(* Logix 5000 project; controller Tekno_ASRS vendor 1 type 14 code 147 rev 20.11; software revision 20.01; part 4 of 4 *)
(* tags used below, declared in another part *)
   AutoMode : BOOL;
   AAxis : AXIS_CIP_DRIVE;
   AAxisMAM : MOTION_INSTRUCTION;
   AAxisMove : BOOL;
   ABGrid : Position[100,20];
   ACompare : REAL;
   AftAreaRest : ALIAS FOR ShuttleIO:8:O.Pt05Data;
   AftAreaScanner : DCI_STOP;
   AftAreaZn1 : ALIAS FOR ShuttleIO:8:O.Pt07Data;
   AftAreaZn4 : ALIAS FOR ShuttleIO:8:O.Pt06Data;
   AftEndZn : BOOL;
   AGVDP : BOOL;
   AGVLightCurtains : DCI_STOP;
   AGVPU : BOOL;
   APos : REAL;
   AReq : DINT;
   ASRSEnable : BOOL;
   AutoConfig : Configuration;
   AxisEnabled : BOOL;
   BAxis : AXIS_CIP_DRIVE;
   BAxisMAM : MOTION_INSTRUCTION;
   BAxisMove : BOOL;
   BCompare : REAL;
   BlowerTm : TIMER;
   BPos : REAL;
   BReq : DINT;
   CommandReq : DINT;
   Configuration : Configuration;
   CReq : DINT;
   CurrentTask : Task;
   DepositReq : BOOL;
   DisableScanners : BOOL;
   DrivesOn : BOOL;
   EStop_SafetyGate : DCI_STOP;
   FootSwitch : ALIAS FOR ShuttleIO:9:I.Pt04Data;
   ForeAreaRst : ALIAS FOR ShuttleIO:8:O.Pt00Data;
   ForeAreaScanner : DCI_STOP;
   ForeAreaZn1 : ALIAS FOR ShuttleIO:8:O.Pt02Data;
   ForeAreaZn4 : ALIAS FOR ShuttleIO:8:O.Pt03Data;
   FwdEndZn : BOOL;
   GZReset : BOOL;
   HighSpdFwd : BOOL;
   HighSpdRev : BOOL;
   JogAct : BOOL;
   LiftStrnOK : BOOL;
   LightCur1 : ALIAS FOR StationaryIO:7:I.Pt06Data;
   LightCur2 : ALIAS FOR StationaryIO:7:I.Pt07Data;
   LightCurEN : ALIAS FOR StationaryIO:6:O.Pt07Data;
   ManConfig : Configuration;
   ManGateClosed : ALIAS FOR ShuttleIO:9:I.Pt02Data;
   MasterReset : BOOL;
   MoveRequested : BOOL;
   OperatorDN : BOOL;
   PalmButtonLeft : ALIAS FOR ShuttleIO:9:I.Pt07Data;
   PalmButtonRight : ALIAS FOR ShuttleIO:9:I.Pt06Data;
   PalmButtons : DCI_STOP;
   PDSimTmr : TIMER;
   ProxPwr : ALIAS FOR StationaryIO:6:O.Pt00Data;
   ResetSafety : BOOL;
   SafetyGate1 : ALIAS FOR StationaryIO:7:I.Pt00Data;
   SafetyGate2 : ALIAS FOR StationaryIO:7:I.Pt01Data;
   SafetyLaserAft1 : ALIAS FOR ShuttleIO:7:I.Pt04Data;
   SafetyLaserAft2 : ALIAS FOR ShuttleIO:7:I.Pt05Data;
   SafetyLaserFore1 : ALIAS FOR ShuttleIO:7:I.Pt00Data;
   SafetyLaserFore2 : ALIAS FOR ShuttleIO:7:I.Pt01Data;
   SafetyResetOns : BOOL;
   StationaryFault : BOOL;
   StationaryHorn : BOOL;
   StationaryManOn : BOOL;
   StationaryRun : BOOL;
   StationaryWarn : BOOL;
   Sts_ASRS_InputsOk : BOOL;
   TaskFIFO : CONTROL;
   TaskFile : Task[100];
   TaskInProcess : BOOL;
   UnBindInProc : BOOL;
   UnBindMotnInProc : BOOL;
   VFDReset : ALIAS FOR ShuttleIO:6:O.Pt00Data;
   XAccuracy : REAL;
   XAxisVFDSS01 : ALIAS FOR ShuttleIO:6:O.Pt04Data;
   XAxisVFDSS02 : ALIAS FOR ShuttleIO:6:O.Pt05Data;
   XHighLimit : REAL;
   XLowLimit : REAL;
   XStrain : Strain;
   XStrainLeftMax : DINT;
   XStrainLeftMin : DINT;
   XStrainRightMax : DINT;
   XStrainRightMin : DINT;
   ZAccuracy : REAL;
   ZADisengage : BOOL;
   ZAftLeftOK : BOOL;
   ZAftRightOK : BOOL;
   ZAftStCalMode : ALIAS FOR ShuttleIO:4:O.Data[0].0;
   ZAftStLftSignRun : ALIAS FOR ShuttleIO:4:I.Data[7].7;
   ZAftStrain : Strain;
   ZAftStrainLeftMax : DINT;
   ZAftStrainLeftMin : DINT;
   ZAftStrainRightMax : DINT;
   ZAftStrainRightMin : DINT;
   ZAftStRtSignRun : ALIAS FOR ShuttleIO:4:I.Data[11].7;
   ZAftStRunMode : ALIAS FOR ShuttleIO:4:O.Data[0].1;
   ZALftTempDint1 : DINT;
   ZALftTempDint2 : DINT;
   ZALftTempFloat1 : REAL;
   ZALftTempFloat2 : REAL;
   ZALftTempFloat3 : REAL;
   ZARgtTempDint1 : DINT;
   ZARgtTempDint2 : DINT;
   ZARgtTempFloat1 : REAL;
   ZARgtTempFloat2 : REAL;
   ZARgtTempFloat3 : REAL;
   ZAxisSafetyDisengage : BOOL;
   ZAxisSafetyLatches : ALIAS FOR ShuttleIO:6:O.Pt07Data;
   ZFLftTempDint1 : DINT;
   ZFLftTempDint2 : DINT;
   ZFLftTempFloat1 : REAL;
   ZFLftTempFloat2 : REAL;
   ZFLftTempFloat3 : REAL;
   ZForeLeftOK : BOOL;
   ZForeRightOK : BOOL;
   ZForeStCalMode : ALIAS FOR ShuttleIO:3:O.Data[0].0;
   ZForeStLftSignRun : ALIAS FOR ShuttleIO:3:I.Data[7].7;
   ZForeStrain : Strain;
   ZForeStrainLeftMax : DINT;
   ZForeStrainLeftMin : DINT;
   ZForeStrainRightMax : DINT;
   ZForeStrainRightMin : DINT;
   ZForeStRtSignRun : ALIAS FOR ShuttleIO:3:I.Data[11].7;
   ZForeStRunMode : ALIAS FOR ShuttleIO:3:O.Data[0].1;
   ZFRgtTempDint1 : DINT;
   ZFRgtTempDint2 : DINT;
   ZFRgtTempFloat1 : REAL;
   ZFRgtTempFloat2 : REAL;
   ZFRgtTempFloat3 : REAL;
   ZHighLimit : REAL;
   ZLBindTmr : TIMER;
   ZLFault : BOOL;
   ZLockMove : MOTION_INSTRUCTION;
   ZLowLimit : REAL;
   ZLProxOK : BOOL;
   ZLReqPosition : REAL;
   ZLRetryDelay : TIMER;
   ZStrainHigh : DINT;
   ZStrainLow : DINT;
(* MainProgram, continued *)

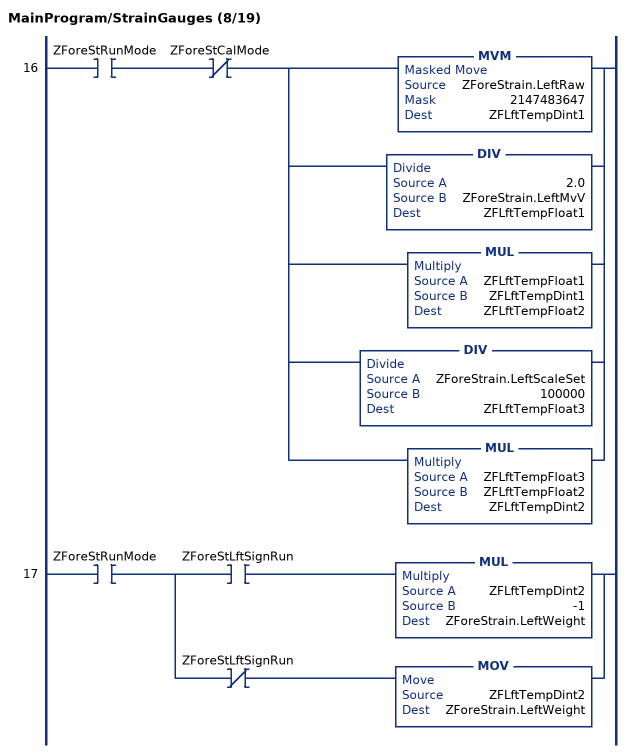
   [picture p48: MainProgram/StrainGauges rungs 16-17]
   16: XIC(ZForeStRunMode)XIO(ZForeStCalMode)[MVM(ZForeStrain.LeftRaw,2147483647,ZFLftTempDint1) ,DIV(2.0,ZForeStrain.LeftMvV,ZFLftTempFloat1) ,MUL(ZFLftTempFloat1,ZFLftTempDint1,ZFLftTempFloat2) ,DIV(ZForeStrain.LeftScaleSet,100000,ZFLftTempFloat3) ,MUL(ZFLftTempFloat3,ZFLftTempFloat2,ZFLftTempDint2) ];
   17: XIC(ZForeStRunMode)[XIC(ZForeStLftSignRun) MUL(ZFLftTempDint2,-1,ZForeStrain.LeftWeight) ,XIO(ZForeStLftSignRun) MOV(ZFLftTempDint2,ZForeStrain.LeftWeight) ];
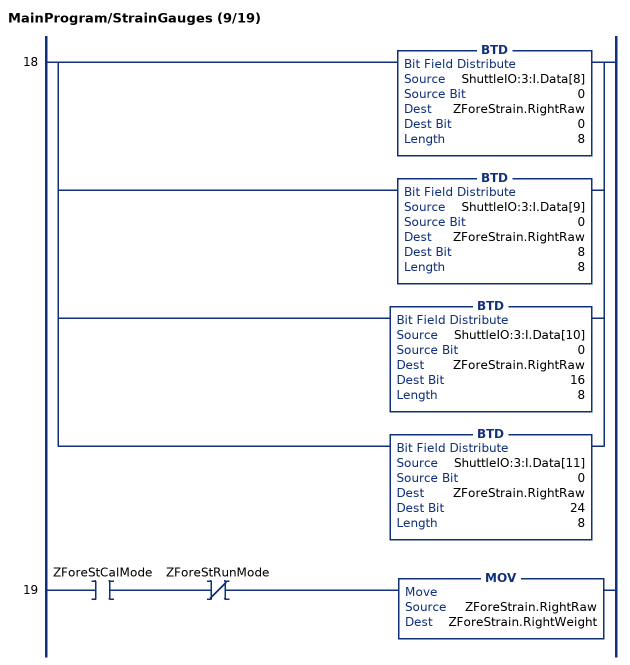
   18: [BTD(ShuttleIO:3:I.Data[8],0,ZForeStrain.RightRaw,0,8) ,BTD(ShuttleIO:3:I.Data[9],0,ZForeStrain.RightRaw,8,8) ,BTD(ShuttleIO:3:I.Data[10],0,ZForeStrain.RightRaw,16,8) ,BTD(ShuttleIO:3:I.Data[11],0,ZForeStrain.RightRaw,24,8) ];
   19: XIC(ZForeStCalMode)XIO(ZForeStRunMode)MOV(ZForeStrain.RightRaw,ZForeStrain.RightWeight);
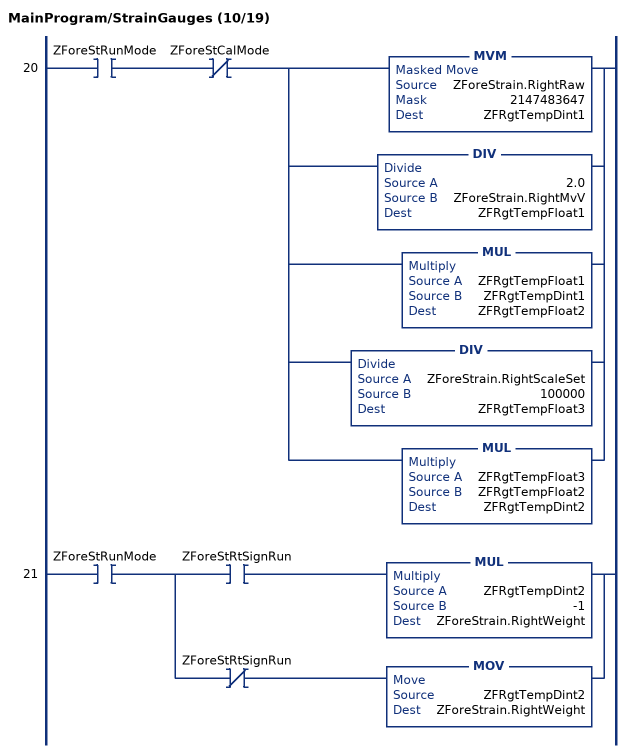
   20: XIC(ZForeStRunMode)XIO(ZForeStCalMode)[MVM(ZForeStrain.RightRaw,2147483647,ZFRgtTempDint1) ,DIV(2.0,ZForeStrain.RightMvV,ZFRgtTempFloat1) ,MUL(ZFRgtTempFloat1,ZFRgtTempDint1,ZFRgtTempFloat2) ,DIV(ZForeStrain.RightScaleSet,100000,ZFRgtTempFloat3) ,MUL(ZFRgtTempFloat3,ZFRgtTempFloat2,ZFRgtTempDint2) ];
   21: XIC(ZForeStRunMode)[XIC(ZForeStRtSignRun) MUL(ZFRgtTempDint2,-1,ZForeStrain.RightWeight) ,XIO(ZForeStRtSignRun) MOV(ZFRgtTempDint2,ZForeStrain.RightWeight) ];
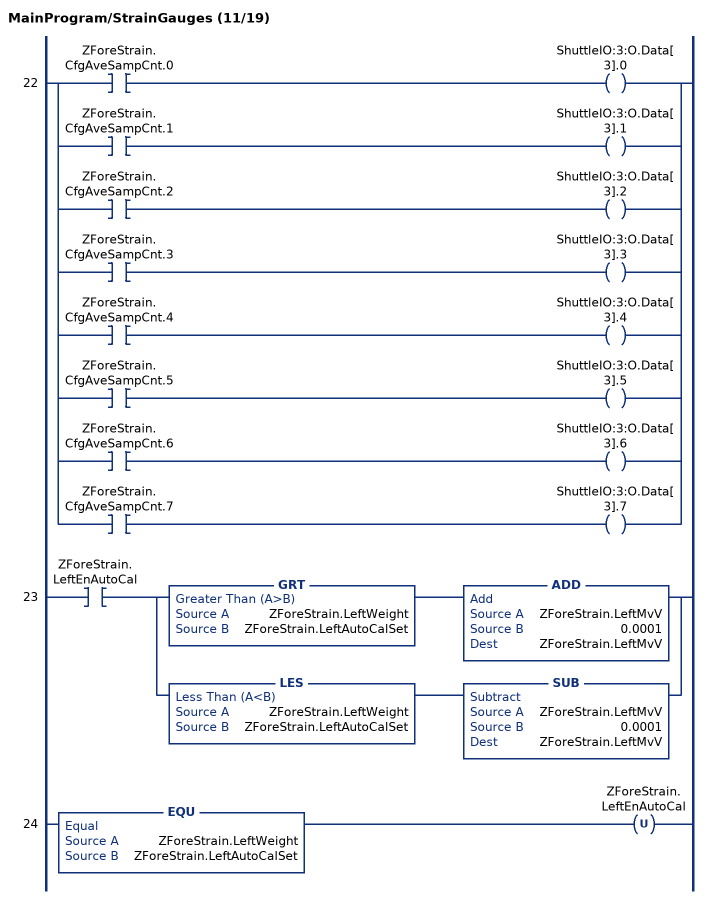
   22: [XIC(ZForeStrain.CfgAveSampCnt.0) OTE(ShuttleIO:3:O.Data[3].0) ,XIC(ZForeStrain.CfgAveSampCnt.1) OTE(ShuttleIO:3:O.Data[3].1) ,XIC(ZForeStrain.CfgAveSampCnt.2) OTE(ShuttleIO:3:O.Data[3].2) ,XIC(ZForeStrain.CfgAveSampCnt.3) OTE(ShuttleIO:3:O.Data[3].3) ,XIC(ZForeStrain.CfgAveSampCnt.4) OTE(ShuttleIO:3:O.Data[3].4) ,XIC(ZForeStrain.CfgAveSampCnt.5) OTE(ShuttleIO:3:O.Data[3].5) ,XIC(ZForeStrain.CfgAveSampCnt.6) OTE(ShuttleIO:3:O.Data[3].6) ,XIC(ZForeStrain.CfgAveSampCnt.7) OTE(ShuttleIO:3:O.Data[3].7) ];
   23: XIC(ZForeStrain.LeftEnAutoCal)[GRT(ZForeStrain.LeftWeight,ZForeStrain.LeftAutoCalSet) ADD(ZForeStrain.LeftMvV,0.0001,ZForeStrain.LeftMvV) ,LES(ZForeStrain.LeftWeight,ZForeStrain.LeftAutoCalSet) SUB(ZForeStrain.LeftMvV,0.0001,ZForeStrain.LeftMvV) ];
   24: EQU(ZForeStrain.LeftWeight,ZForeStrain.LeftAutoCalSet)OTU(ZForeStrain.LeftEnAutoCal);
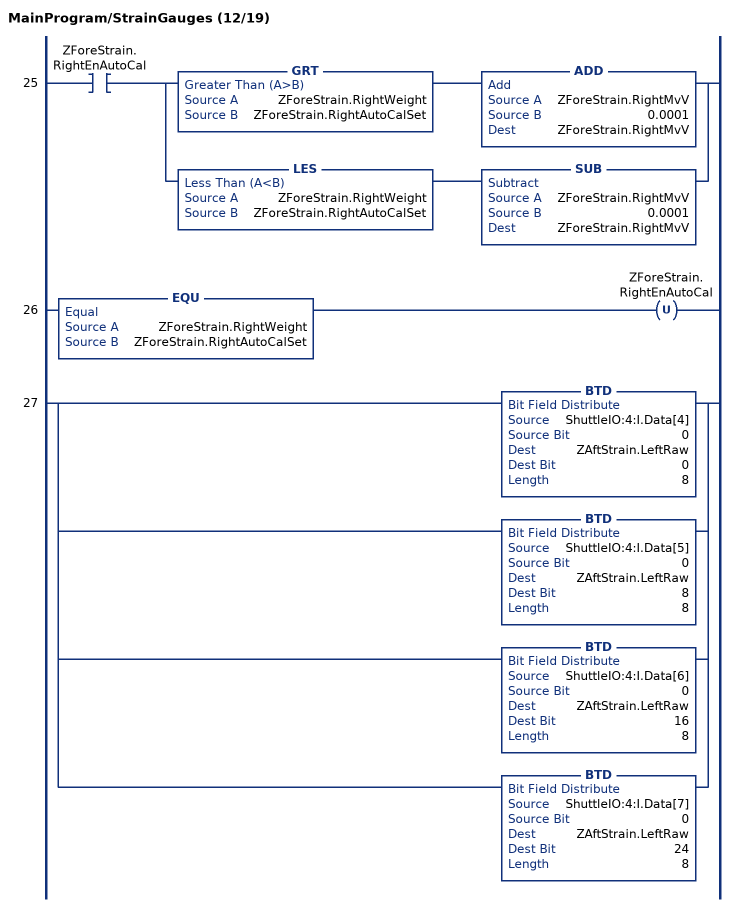
   25: XIC(ZForeStrain.RightEnAutoCal)[GRT(ZForeStrain.RightWeight,ZForeStrain.RightAutoCalSet) ADD(ZForeStrain.RightMvV,0.0001,ZForeStrain.RightMvV) ,LES(ZForeStrain.RightWeight,ZForeStrain.RightAutoCalSet) SUB(ZForeStrain.RightMvV,0.0001,ZForeStrain.RightMvV) ];
   26: EQU(ZForeStrain.RightWeight,ZForeStrain.RightAutoCalSet)OTU(ZForeStrain.RightEnAutoCal);
   27: [BTD(ShuttleIO:4:I.Data[4],0,ZAftStrain.LeftRaw,0,8) ,BTD(ShuttleIO:4:I.Data[5],0,ZAftStrain.LeftRaw,8,8) ,BTD(ShuttleIO:4:I.Data[6],0,ZAftStrain.LeftRaw,16,8) ,BTD(ShuttleIO:4:I.Data[7],0,ZAftStrain.LeftRaw,24,8) ];
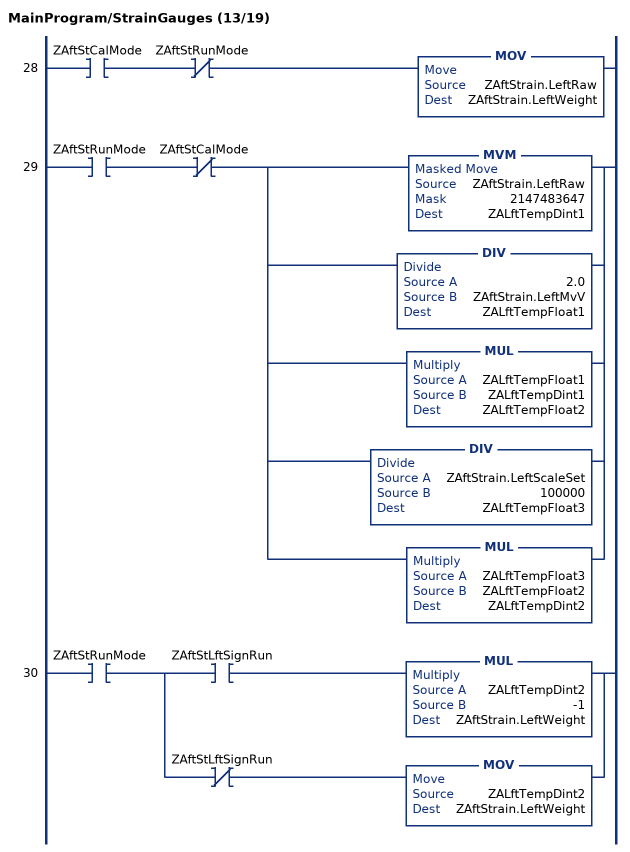
   28: XIC(ZAftStCalMode)XIO(ZAftStRunMode)MOV(ZAftStrain.LeftRaw,ZAftStrain.LeftWeight);
   29: XIC(ZAftStRunMode)XIO(ZAftStCalMode)[MVM(ZAftStrain.LeftRaw,2147483647,ZALftTempDint1) ,DIV(2.0,ZAftStrain.LeftMvV,ZALftTempFloat1) ,MUL(ZALftTempFloat1,ZALftTempDint1,ZALftTempFloat2) ,DIV(ZAftStrain.LeftScaleSet,100000,ZALftTempFloat3) ,MUL(ZALftTempFloat3,ZALftTempFloat2,ZALftTempDint2) ];
   30: XIC(ZAftStRunMode)[XIC(ZAftStLftSignRun) MUL(ZALftTempDint2,-1,ZAftStrain.LeftWeight) ,XIO(ZAftStLftSignRun) MOV(ZALftTempDint2,ZAftStrain.LeftWeight) ];
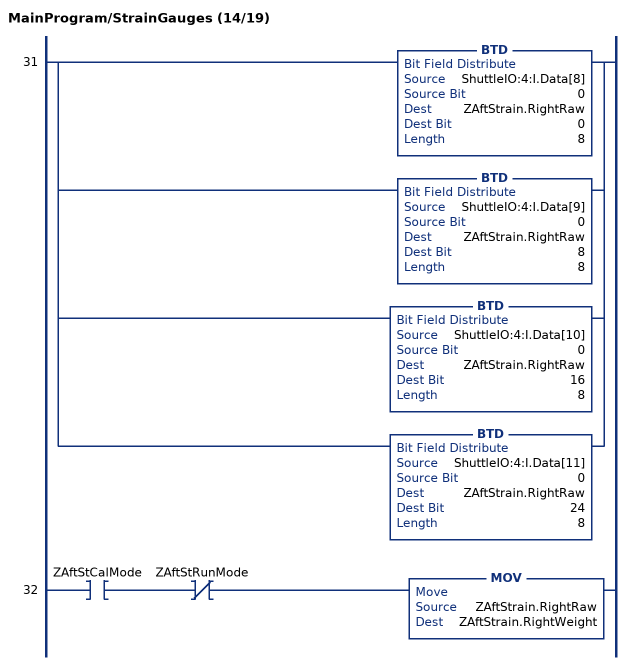
   31: [BTD(ShuttleIO:4:I.Data[8],0,ZAftStrain.RightRaw,0,8) ,BTD(ShuttleIO:4:I.Data[9],0,ZAftStrain.RightRaw,8,8) ,BTD(ShuttleIO:4:I.Data[10],0,ZAftStrain.RightRaw,16,8) ,BTD(ShuttleIO:4:I.Data[11],0,ZAftStrain.RightRaw,24,8) ];
   32: XIC(ZAftStCalMode)XIO(ZAftStRunMode)MOV(ZAftStrain.RightRaw,ZAftStrain.RightWeight);
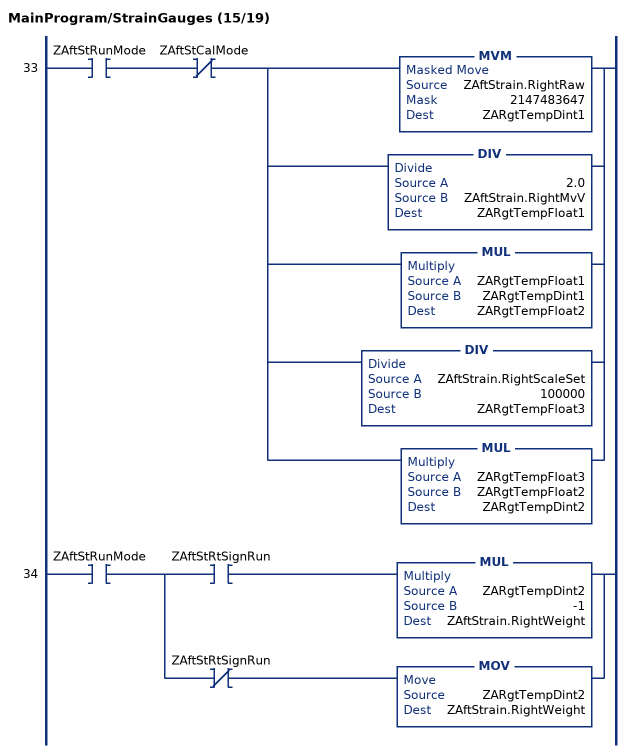
   33: XIC(ZAftStRunMode)XIO(ZAftStCalMode)[MVM(ZAftStrain.RightRaw,2147483647,ZARgtTempDint1) ,DIV(2.0,ZAftStrain.RightMvV,ZARgtTempFloat1) ,MUL(ZARgtTempFloat1,ZARgtTempDint1,ZARgtTempFloat2) ,DIV(ZAftStrain.RightScaleSet,100000,ZARgtTempFloat3) ,MUL(ZARgtTempFloat3,ZARgtTempFloat2,ZARgtTempDint2) ];
   34: XIC(ZAftStRunMode)[XIC(ZAftStRtSignRun) MUL(ZARgtTempDint2,-1,ZAftStrain.RightWeight) ,XIO(ZAftStRtSignRun) MOV(ZARgtTempDint2,ZAftStrain.RightWeight) ];
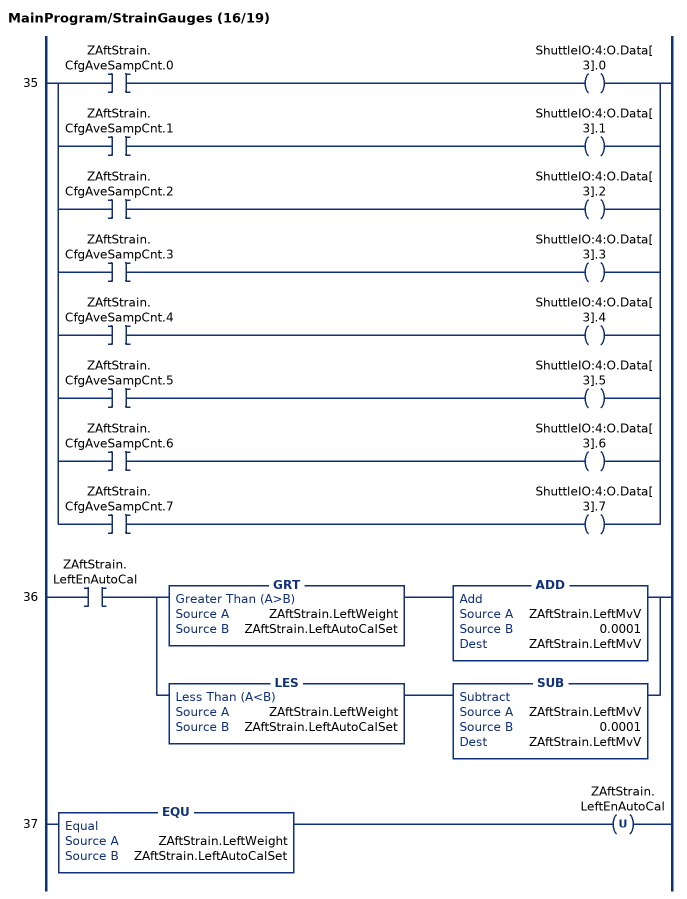
   35: [XIC(ZAftStrain.CfgAveSampCnt.0) OTE(ShuttleIO:4:O.Data[3].0) ,XIC(ZAftStrain.CfgAveSampCnt.1) OTE(ShuttleIO:4:O.Data[3].1) ,XIC(ZAftStrain.CfgAveSampCnt.2) OTE(ShuttleIO:4:O.Data[3].2) ,XIC(ZAftStrain.CfgAveSampCnt.3) OTE(ShuttleIO:4:O.Data[3].3) ,XIC(ZAftStrain.CfgAveSampCnt.4) OTE(ShuttleIO:4:O.Data[3].4) ,XIC(ZAftStrain.CfgAveSampCnt.5) OTE(ShuttleIO:4:O.Data[3].5) ,XIC(ZAftStrain.CfgAveSampCnt.6) OTE(ShuttleIO:4:O.Data[3].6) ,XIC(ZAftStrain.CfgAveSampCnt.7) OTE(ShuttleIO:4:O.Data[3].7) ];
   36: XIC(ZAftStrain.LeftEnAutoCal)[GRT(ZAftStrain.LeftWeight,ZAftStrain.LeftAutoCalSet) ADD(ZAftStrain.LeftMvV,0.0001,ZAftStrain.LeftMvV) ,LES(ZAftStrain.LeftWeight,ZAftStrain.LeftAutoCalSet) SUB(ZAftStrain.LeftMvV,0.0001,ZAftStrain.LeftMvV) ];
   37: EQU(ZAftStrain.LeftWeight,ZAftStrain.LeftAutoCalSet)OTU(ZAftStrain.LeftEnAutoCal);
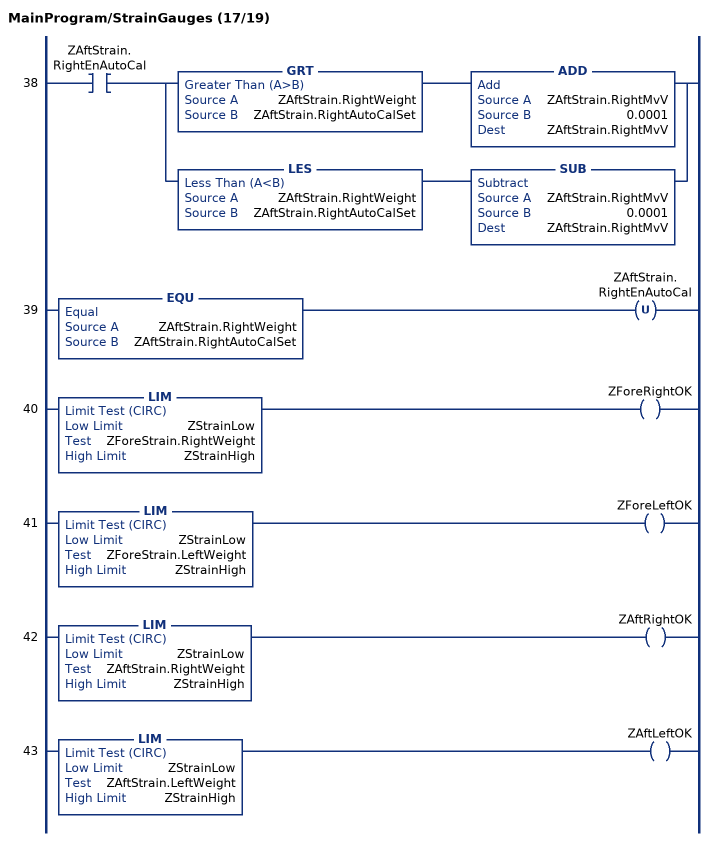
   38: XIC(ZAftStrain.RightEnAutoCal)[GRT(ZAftStrain.RightWeight,ZAftStrain.RightAutoCalSet) ADD(ZAftStrain.RightMvV,0.0001,ZAftStrain.RightMvV) ,LES(ZAftStrain.RightWeight,ZAftStrain.RightAutoCalSet) SUB(ZAftStrain.RightMvV,0.0001,ZAftStrain.RightMvV) ];
   39: EQU(ZAftStrain.RightWeight,ZAftStrain.RightAutoCalSet)OTU(ZAftStrain.RightEnAutoCal);
   40: LIM(ZStrainLow,ZForeStrain.RightWeight,ZStrainHigh)OTE(ZForeRightOK);
   41: LIM(ZStrainLow,ZForeStrain.LeftWeight,ZStrainHigh)OTE(ZForeLeftOK);
   42: LIM(ZStrainLow,ZAftStrain.RightWeight,ZStrainHigh)OTE(ZAftRightOK);
   43: LIM(ZStrainLow,ZAftStrain.LeftWeight,ZStrainHigh)OTE(ZAftLeftOK);
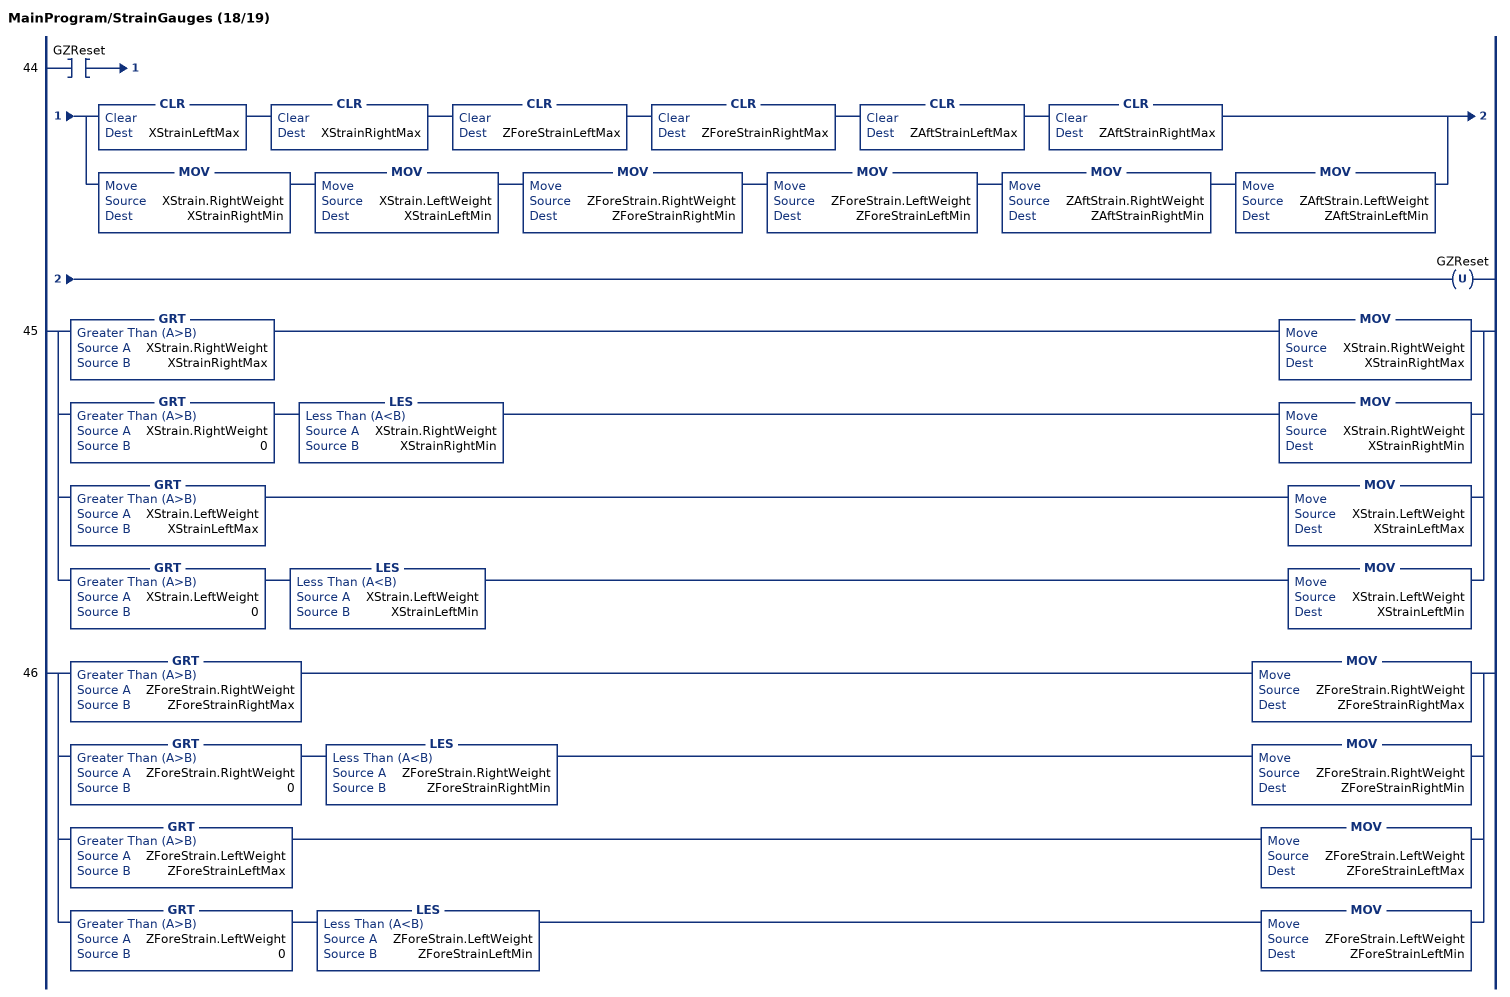
   44: XIC(GZReset)[CLR(XStrainLeftMax) CLR(XStrainRightMax) CLR(ZForeStrainLeftMax) CLR(ZForeStrainRightMax) CLR(ZAftStrainLeftMax) CLR(ZAftStrainRightMax) ,MOV(XStrain.RightWeight,XStrainRightMin) MOV(XStrain.LeftWeight,XStrainLeftMin) MOV(ZForeStrain.RightWeight,ZForeStrainRightMin) MOV(ZForeStrain.LeftWeight,ZForeStrainLeftMin) MOV(ZAftStrain.RightWeight,ZAftStrainRightMin) MOV(ZAftStrain.LeftWeight,ZAftStrainLeftMin) ]OTU(GZReset);
   45: [GRT(XStrain.RightWeight,XStrainRightMax) MOV(XStrain.RightWeight,XStrainRightMax) ,GRT(XStrain.RightWeight,0) LES(XStrain.RightWeight,XStrainRightMin) MOV(XStrain.RightWeight,XStrainRightMin) ,GRT(XStrain.LeftWeight,XStrainLeftMax) MOV(XStrain.LeftWeight,XStrainLeftMax) ,GRT(XStrain.LeftWeight,0) LES(XStrain.LeftWeight,XStrainLeftMin) MOV(XStrain.LeftWeight,XStrainLeftMin) ];
   46: [GRT(ZForeStrain.RightWeight,ZForeStrainRightMax) MOV(ZForeStrain.RightWeight,ZForeStrainRightMax) ,GRT(ZForeStrain.RightWeight,0) LES(ZForeStrain.RightWeight,ZForeStrainRightMin) MOV(ZForeStrain.RightWeight,ZForeStrainRightMin) ,GRT(ZForeStrain.LeftWeight,ZForeStrainLeftMax) MOV(ZForeStrain.LeftWeight,ZForeStrainLeftMax) ,GRT(ZForeStrain.LeftWeight,0) LES(ZForeStrain.LeftWeight,ZForeStrainLeftMin) MOV(ZForeStrain.LeftWeight,ZForeStrainLeftMin) ];
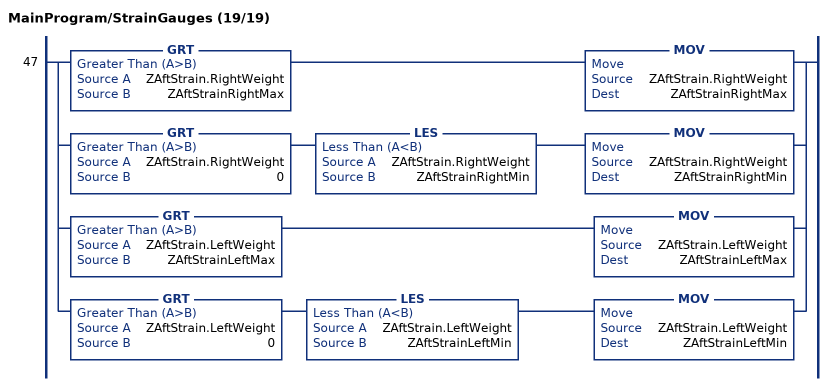
   47: [GRT(ZAftStrain.RightWeight,ZAftStrainRightMax) MOV(ZAftStrain.RightWeight,ZAftStrainRightMax) ,GRT(ZAftStrain.RightWeight,0) LES(ZAftStrain.RightWeight,ZAftStrainRightMin) MOV(ZAftStrain.RightWeight,ZAftStrainRightMin) ,GRT(ZAftStrain.LeftWeight,ZAftStrainLeftMax) MOV(ZAftStrain.LeftWeight,ZAftStrainLeftMax) ,GRT(ZAftStrain.LeftWeight,0) LES(ZAftStrain.LeftWeight,ZAftStrainLeftMin) MOV(ZAftStrain.LeftWeight,ZAftStrainLeftMin) ];
END_ROUTINE

ROUTINE Task_List_Processor   (* ladder *)
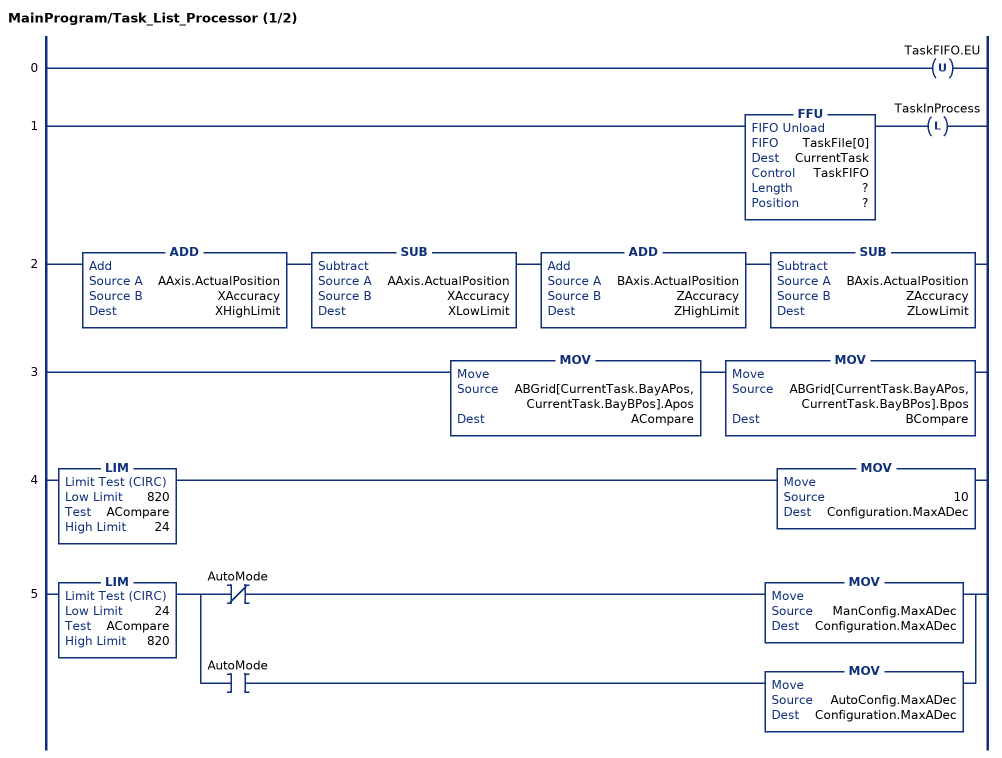
   0: OTU(TaskFIFO.EU);
   1: FFU(TaskFile[0],CurrentTask,TaskFIFO,?,?)OTL(TaskInProcess);
   2: ADD(AAxis.ActualPosition,XAccuracy,XHighLimit)SUB(AAxis.ActualPosition,XAccuracy,XLowLimit)ADD(BAxis.ActualPosition,ZAccuracy,ZHighLimit)SUB(BAxis.ActualPosition,ZAccuracy,ZLowLimit);
   3: MOV(ABGrid[CurrentTask.BayAPos,CurrentTask.BayBPos].Apos,ACompare)MOV(ABGrid[CurrentTask.BayAPos,CurrentTask.BayBPos].Bpos,BCompare);
   4: LIM(820,ACompare,24)MOV(10,Configuration.MaxADec);
   5: LIM(24,ACompare,820)[XIO(AutoMode) MOV(ManConfig.MaxADec,Configuration.MaxADec) ,XIC(AutoMode) MOV(AutoConfig.MaxADec,Configuration.MaxADec) ];
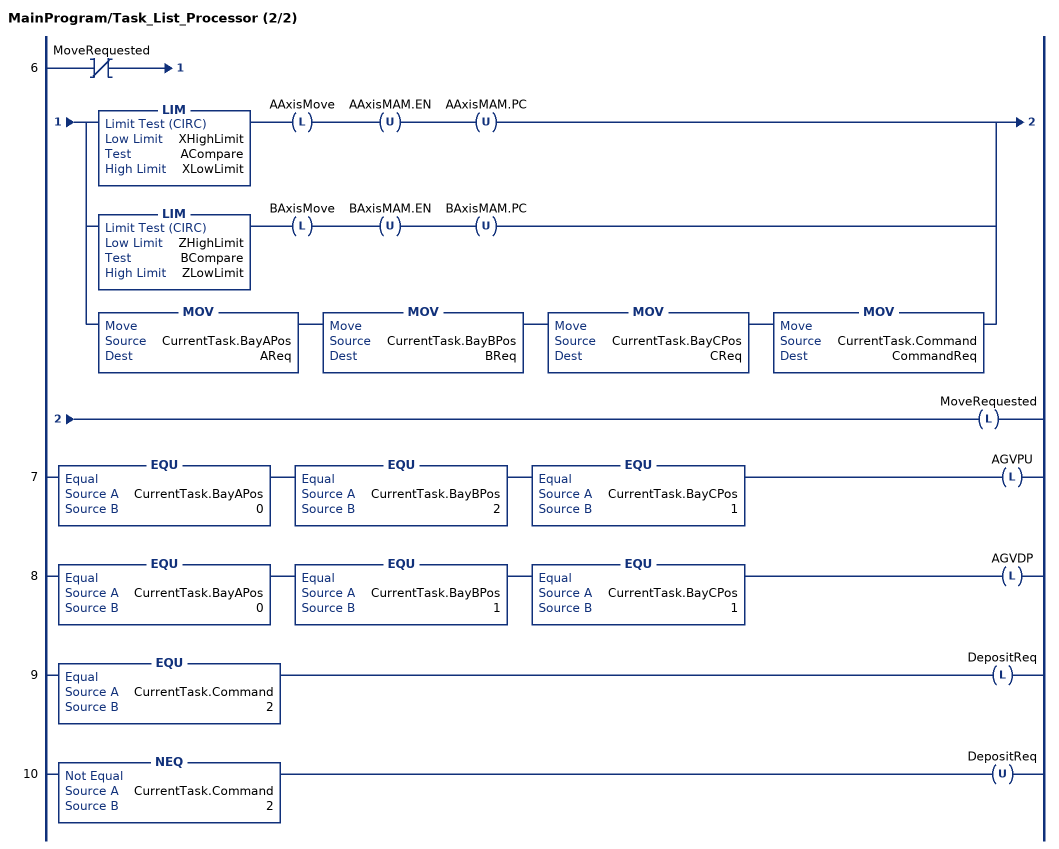
   6: XIO(MoveRequested)[LIM(XHighLimit,ACompare,XLowLimit) OTL(AAxisMove) OTU(AAxisMAM.EN) OTU(AAxisMAM.PC) ,LIM(ZHighLimit,BCompare,ZLowLimit) OTL(BAxisMove) OTU(BAxisMAM.EN) OTU(BAxisMAM.PC) ,MOV(CurrentTask.BayAPos,AReq) MOV(CurrentTask.BayBPos,BReq) MOV(CurrentTask.BayCPos,CReq) MOV(CurrentTask.Command,CommandReq) ]OTL(MoveRequested);
   7: EQU(CurrentTask.BayAPos,0)EQU(CurrentTask.BayBPos,2)EQU(CurrentTask.BayCPos,1)OTL(AGVPU);
   8: EQU(CurrentTask.BayAPos,0)EQU(CurrentTask.BayBPos,1)EQU(CurrentTask.BayCPos,1)OTL(AGVDP);
   9: EQU(CurrentTask.Command,2)OTL(DepositReq);
   10: NEQ(CurrentTask.Command,2)OTU(DepositReq);
END_ROUTINE

ROUTINE VisitPorD   (* ladder *)
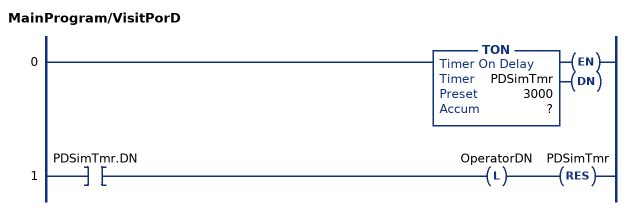
   0: TON(PDSimTmr,?,?);
   1: XIC(PDSimTmr.DN)OTL(OperatorDN)RES(PDSimTmr);
END_ROUTINE

ROUTINE ZLock_Release   (* ladder *)
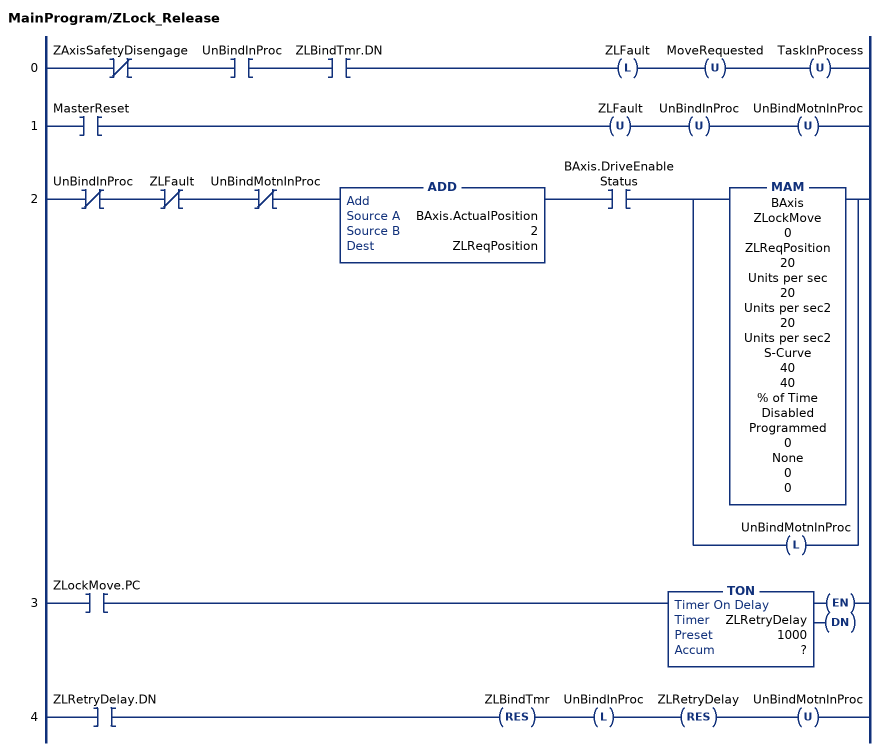
   0: XIO(ZAxisSafetyDisengage)XIC(UnBindInProc)XIC(ZLBindTmr.DN)OTL(ZLFault)OTU(MoveRequested)OTU(TaskInProcess);
   1: XIC(MasterReset)OTU(ZLFault)OTU(UnBindInProc)OTU(UnBindMotnInProc);
   2: XIO(UnBindInProc)XIO(ZLFault)XIO(UnBindMotnInProc)ADD(BAxis.ActualPosition,2,ZLReqPosition)XIC(BAxis.DriveEnableStatus)[MAM(BAxis,ZLockMove,0,ZLReqPosition,20,Units per sec,20,Units per sec2,20,Units per sec2,S-Curve,40,40,% of Time,Disabled,Programmed,0,None,0,0) ,OTL(UnBindMotnInProc) ];
   3: XIC(ZLockMove.PC)TON(ZLRetryDelay,?,?);
   4: XIC(ZLRetryDelay.DN)RES(ZLBindTmr)OTL(UnBindInProc)RES(ZLRetryDelay)OTU(UnBindMotnInProc);
END_ROUTINE
END_PROGRAM

PROGRAM SafetyProgram   (* main routine MainRoutine *)
VAR
   alkjdfl : BOOL;
   Lift : DINT;
   ljfalsj : BOOL;
END_VAR

ROUTINE MainRoutine   (* ladder *)
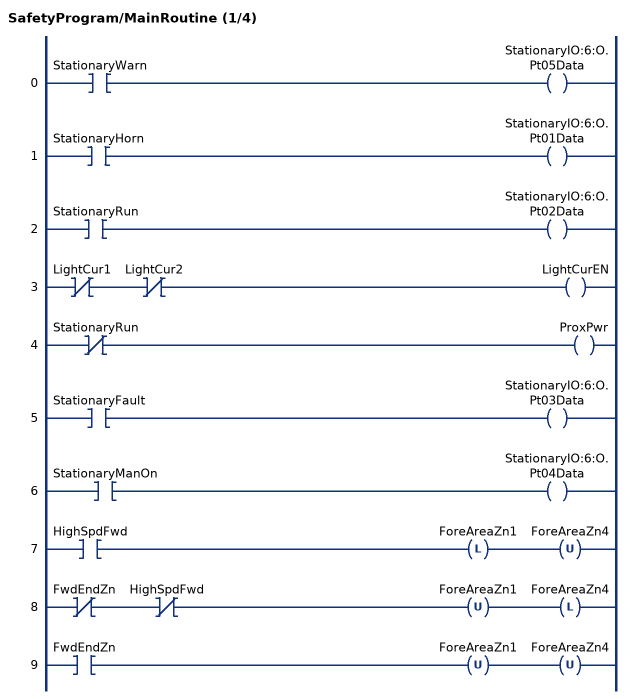
   0: XIC(StationaryWarn)OTE(StationaryIO:6:O.Pt05Data);
   1: XIC(StationaryHorn)OTE(StationaryIO:6:O.Pt01Data);
   2: XIC(StationaryRun)OTE(StationaryIO:6:O.Pt02Data);
   3: XIO(LightCur1)XIO(LightCur2)OTE(LightCurEN);
   4: XIO(StationaryRun)OTE(ProxPwr);
   5: XIC(StationaryFault)OTE(StationaryIO:6:O.Pt03Data);
   6: XIC(StationaryManOn)OTE(StationaryIO:6:O.Pt04Data);
   7: XIC(HighSpdFwd)OTL(ForeAreaZn1)OTU(ForeAreaZn4);
   8: XIO(FwdEndZn)XIO(HighSpdFwd)OTU(ForeAreaZn1)OTL(ForeAreaZn4);
   9: XIC(FwdEndZn)OTU(ForeAreaZn1)OTU(ForeAreaZn4);
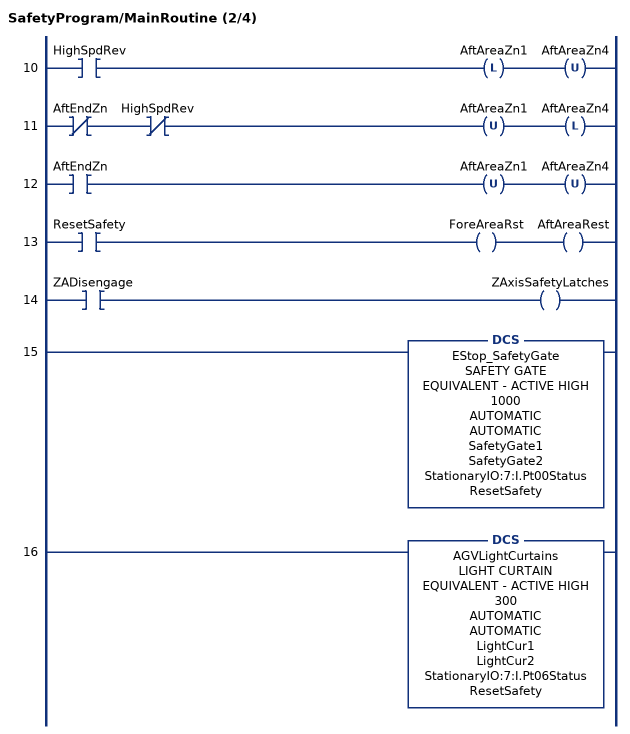
   10: XIC(HighSpdRev)OTL(AftAreaZn1)OTU(AftAreaZn4);
   11: XIO(AftEndZn)XIO(HighSpdRev)OTU(AftAreaZn1)OTL(AftAreaZn4);
   12: XIC(AftEndZn)OTU(AftAreaZn1)OTU(AftAreaZn4);
   13: XIC(ResetSafety)OTE(ForeAreaRst)OTE(AftAreaRest);
   14: XIC(ZADisengage)OTE(ZAxisSafetyLatches);
   15: DCS(EStop_SafetyGate,SAFETY GATE,EQUIVALENT - ACTIVE HIGH,1000,AUTOMATIC,AUTOMATIC,SafetyGate1,SafetyGate2,StationaryIO:7:I.Pt00Status,ResetSafety);
   16: DCS(AGVLightCurtains,LIGHT CURTAIN,EQUIVALENT - ACTIVE HIGH,300,AUTOMATIC,AUTOMATIC,LightCur1,LightCur2,StationaryIO:7:I.Pt06Status,ResetSafety);
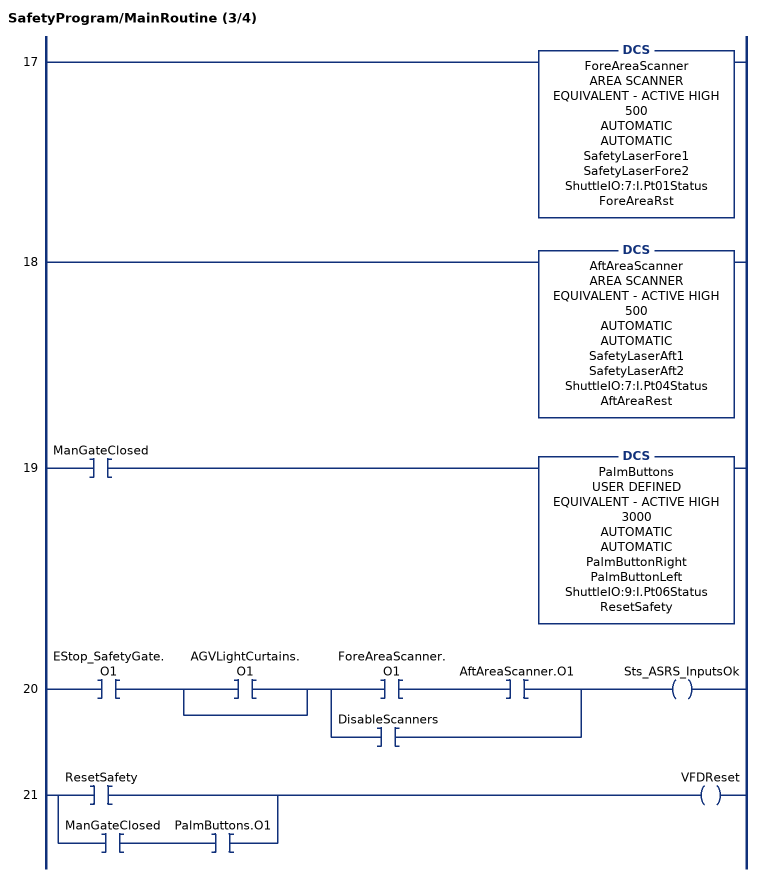
   17: DCS(ForeAreaScanner,AREA SCANNER,EQUIVALENT - ACTIVE HIGH,500,AUTOMATIC,AUTOMATIC,SafetyLaserFore1,SafetyLaserFore2,ShuttleIO:7:I.Pt01Status,ForeAreaRst);
   18: DCS(AftAreaScanner,AREA SCANNER,EQUIVALENT - ACTIVE HIGH,500,AUTOMATIC,AUTOMATIC,SafetyLaserAft1,SafetyLaserAft2,ShuttleIO:7:I.Pt04Status,AftAreaRest);
   19: XIC(ManGateClosed)DCS(PalmButtons,USER DEFINED,EQUIVALENT - ACTIVE HIGH,3000,AUTOMATIC,AUTOMATIC,PalmButtonRight,PalmButtonLeft,ShuttleIO:9:I.Pt06Status,ResetSafety);
   20: XIC(EStop_SafetyGate.O1)[XIC(AGVLightCurtains.O1) ,][XIC(ForeAreaScanner.O1) XIC(AftAreaScanner.O1) ,XIC(DisableScanners) ]OTE(Sts_ASRS_InputsOk);
   21: [XIC(ResetSafety) ,XIC(ManGateClosed) XIC(PalmButtons.O1) ]OTE(VFDReset);
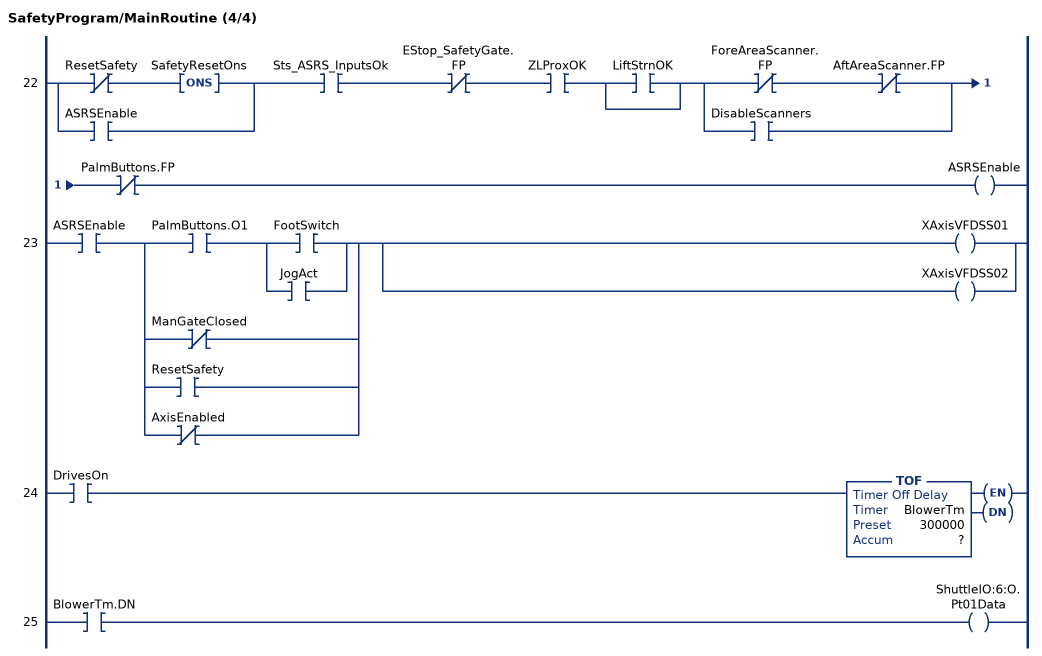
   22: [XIO(ResetSafety) ONS(SafetyResetOns) ,XIC(ASRSEnable) ]XIC(Sts_ASRS_InputsOk)XIO(EStop_SafetyGate.FP)XIC(ZLProxOK)[XIC(LiftStrnOK) ,][XIO(ForeAreaScanner.FP) XIO(AftAreaScanner.FP) ,XIC(DisableScanners) ]XIO(PalmButtons.FP)OTE(ASRSEnable);
   23: XIC(ASRSEnable)[XIC(PalmButtons.O1) [XIC(FootSwitch) ,XIC(JogAct) ] ,XIO(ManGateClosed) ,XIC(ResetSafety) ,XIO(AxisEnabled) ][OTE(XAxisVFDSS01) ,OTE(XAxisVFDSS02) ];
   24: XIC(DrivesOn)TOF(BlowerTm,?,?);
   25: XIC(BlowerTm.DN)OTE(ShuttleIO:6:O.Pt01Data);
END_ROUTINE
END_PROGRAM
